{attribute 'GeneratedUsingTerminal: EK1100-0000-0018'}
{attribute addProperty BoxType "EK1100-0000-0018"}
{attribute addProperty Id "Beckhoff_EPP6xxxEK1122Beckhoff_EPP6xxxEK1122_92E40431672"}
{attribute addProperty CRC "3750280943"}
{attribute addProperty Size "672"}
TYPE Beckhoff_EPP6xxx_DF88BEEF EXTENDS EK1100_AB5A9467 :
STRUCT
	{attribute addProperty Name "Beckhoff_EPP6xxxEK1122"}
	{attribute addProperty PreviousPort "Beckhoff EPP6xxx : B"}
	Beckhoff_EPP6xxxEK1122 : Beckhoff_EPP6xxxEK1122_92E40431;
END_STRUCT
END_TYPE

(* stored: Version 1.2.0.0, ProductVersion 3.1.4024.9
   DUT Beckhoff_EPP6xxx_DF88BEEF: Id {a1119d5c-322b-48f4-bc23-5663b0360d87} *)
